TYPE AlternativeOperation :
STRUCT
	EN: BOOL;
	Polarity: BOOL;
	ActivateViaDI: BOOL;
	ActivateViaADS: BOOL;
	SPTemperature: LREAL;
	UseSPTemperature: BOOL;
	SPSupplyAirPressure: LREAL;
	SPExtractAirPressure: LREAL;
	SPSupplyAirFlow: LREAL;
	SPExtractAirFlow: LREAL;
	StopUnit: BOOL;
	UnitOperation: UnitOperation;
END_STRUCT
END_TYPE

(* stored: Version 1.1.0.1, ProductVersion 3.1.4024.6
   DUT AlternativeOperation: Id {84b3bb15-5ec5-4e46-b08a-b20e6c2e92cd} *)
